(* IEC 61131-3 sources: test_fernando/Modicon_M660C.device.xml.v3^/Plc Logic.plclogic.xml.v3^/Application.application.xml.v3^/RealTimeClock/SR_RealTimeClock.prg.st^, 4 files *)

(* ---- ldtLocalTime.prop.st ---- *)
 {attribute 'monitoring':='variable'}
PROPERTY ldtLocalTime : LDATE_AND_TIME //If local time is not supported, the return value is 0 (LDT#1970-1-1-0:0:0)
__GETTERDECLARATION__
VAR
	uliTimestamp : ULINT;
	stDate: SysTimeRtc.SYSTIMEDATE;
END_VAR
__GETTERIMPLEMENTATION__
//Get RTC from PLC
uliTimestamp := TO_ULINT(ldtRtc)/1000000;

IF udiLastResultGetRtc <> CmpErrors.Errors.ERR_OK THEN
	RETURN;
END_IF

//Convert RTC to local time
uidLastResultLocalTimeConvertToLocal := SysTimeRtc.SysTimeRtcConvertHighResToLocal(pTimestamp := uliTimestamp, pDate := stDate);

IF uidLastResultLocalTimeConvertToLocal <> CmpErrors.Errors.ERR_OK THEN
	RETURN;
END_IF

uidLastResultLocalTimeConvertToHighRes := SysTimeRtc.SysTimeRtcConvertDateToHighRes(pDate := stDate, pTimestamp := uliTimestamp);

IF uidLastResultLocalTimeConvertToHighRes <> CmpErrors.Errors.ERR_OK THEN
	RETURN;
END_IF

//Return as LDT
ldtLocalTime := TO_LDT(uliTimestamp*1000000);

(* ---- ldtRtc.prop.st ---- *)
 {attribute 'monitoring':='variable'}
PROPERTY ldtRtc : LDATE_AND_TIME
__GETTERDECLARATION__
VAR
	uliRtc: ULINT;
END_VAR
__GETTERIMPLEMENTATION__
//Get RTC from PLC
udiLastResultGetRtc := SysTimeRtc.SysTimeRtcHighResGet(pTimestamp := uliRtc);

IF udiLastResultGetRtc <> CmpErrors.Errors.ERR_OK THEN
	RETURN;
END_IF

//Return as LDT
ldtRtc := TO_LDT(uliRtc*1000000);

(* ---- SetRtc.meth.st ---- *)
/// This method is used to set the RealTimeClock of the controller.

METHOD SetRtc
VAR_INPUT
	i_ldtTimestamp : LDATE_AND_TIME; //Timestamp to set
	i_xWriteAsUtc    : BOOL := TRUE; //If TRUE the timestamp is converted to UTC before writing, else it is written as it is to the RTC.
END_VAR
VAR_OUTPUT
	q_xError     : BOOL; //Indicates that an error was detected during execution
	q_udiResult  : SysTimeRtc.SysTypes.RTS_IEC_RESULT; // Provides diagnostic and status information as a numeric value
	q_sResultMsg : STRING; //Provides additional diagnostic and status information as a text message
END_VAR
VAR
	udiResult  : SysTimeRtc.SysTypes.RTS_IEC_RESULT;

	uliTimestamp : ULINT;
	stDate       : SysTimeRtc.SYSTIMEDATE;
END_VAR

//Convert LDT to ULINT
uliTimestamp := TO_ULINT(i_ldtTimestamp)/1000000;

IF i_xWriteAsUtc THEN
	//Convert timestamp to local time
	udiResult := SysTimeRtc.SysTimeRtcConvertHighResToDate(pTimestamp := uliTimestamp, pDate := stDate);

	IF udiResult <> CmpErrors.Errors.ERR_OK THEN
		q_xError := TRUE;
		q_udiResult := udiResult;
		q_sResultMsg := CONCAT('Function SysTimeRtcConvertHighResToDate failed with result ', TO_STRING(udiResult));
		RETURN;
	END_IF

	udiResult := SysTimeRtc.SysTimeRtcConvertLocalToHighRes(pDate := stDate, pTimestamp := uliTimestamp);

	IF udiResult <> CmpErrors.Errors.ERR_OK THEN
		q_xError := TRUE;
		q_udiResult := udiResult;
		q_sResultMsg := CONCAT('Function SysTimeRtcConvertLocalToHighRes failed with result ', TO_STRING(udiResult));
		RETURN;
	END_IF

END_IF

//Set RTC to PLC
udiResult := SysTimeRtc.SysTimeRtcHighResSet(pTimestamp := uliTimestamp);

//Set outputs
IF udiResult <> CmpErrors.Errors.ERR_OK THEN
	q_xError := TRUE;
	q_udiResult := udiResult;
	q_sResultMsg := CONCAT('Function SysTimeRtc failed with result ', TO_STRING(udiResult));
	RETURN;
END_IF

q_xError := FALSE;
q_udiResult := CmpErrors.Errors.ERR_OK;
q_sResultMsg := 'RTC successfully set';

(* ---- stTimezone.prop.st ---- *)
 {attribute 'monitoring':='variable'}
PROPERTY stTimezone : REFERENCE TO SysTimeRtc.TimezoneInformation2; //If utcOffsetSeconds is not supported, the return value of this structure element is -1
__GETTERDECLARATION__
VAR
END_VAR
__GETTERIMPLEMENTATION__
//Get timezone from PLC
udiLastResultGetTimezone := SysTimeRtc.SysTimeRtcGetTimezone2(pTZI := stTimezone_loc);

IF udiLastResultGetTimezone <> CmpErrors.Errors.ERR_OK THEN
	RETURN;
END_IF

stTimezone REF= stTimezone_loc;
